FUNCTION_BLOCK MNG_Simulation
VAR_INPUT
    bEnable    : BOOL                          := FALSE;
    outputs AT %I*   : MNG_Application_Outputs_32Bit         ;
END_VAR
VAR_OUTPUT
    inputs AT %Q*  : MNG_Application_Inputs_32Bit          ;
END_VAR
VAR
    ioUpdater  : MNG_UpdateIOs                 := (sRemoteHost := '192.168.42.31', nRemotePort := 7000);
    fbCloseAll : FB_SocketCloseAll;
    bCloseAll  : BOOL := TRUE;
END_VAR

(* @END_DECLARATION := '0'                                                    *)
IF bCloseAll THEN (*On PLC reset or program download close all old (opened) connections *)
    bCloseAll := FALSE;
    fbCloseAll( bExecute:= TRUE );
ELSE
    fbCloseAll( bExecute:= FALSE );
END_IF

IF NOT fbCloseAll.bBusy THEN

    (* ------------------------------------- trigger data exchange ----------------------------------------------------------------------------*)
    ioUpdater(Outputs := outputs, Inputs := inputs, bEnable := bEnable);

END_IF

END_FUNCTION_BLOCK

(* stored: Version 1.1.0.1, ProductVersion 3.1.0.23 *)
